FUNCTION_BLOCK FB_Stop
VAR_INPUT
(*È«¾Ö*)
	Mode:DINT;
	PowerState:BOOL;
	CoupleState:DINT;
	(*GapMode*)
	GapStop:BOOL;
	(*BCGapMode*)
	BCGapStop:BOOL;
	(*SingleCarrierMode*)
	TopStop:BOOL;
	BottomStop:BOOL;
	InStop:BOOL;
	OutStop:BOOL;
	(*DebugMode*)
	LeftTopStop:BOOL;
	RightTopStop:BOOL;
	LeftBottomStop:BOOL;
	RightBottomStop:BOOL;
	LeftInStop:BOOL;
	RightInStop:BOOL;
	LeftOutStop:BOOL;
	RightOutStop:BOOL;
END_VAR
VAR_OUTPUT
	FbID:DINT:=1001;
	GapState:DINT;
	GapBusy:BOOL;
	GapDone:BOOL;

	BCGapState:DINT;
	BCGapBusy:BOOL;
	BCGapDone:BOOL;

	TopState:DINT;
	TopBusy:BOOL;
	TopDone:BOOL;
	BottomState:DINT;
	BottomBusy:BOOL;
	BottomDone:BOOL;
	InState:DINT;
	InBusy:BOOL;
	InDone:BOOL;
	OutState:DINT;
	OutBusy:BOOL;
	OutDone:BOOL;

	LeftTopState:DINT;
	LeftTopBusy:BOOL;
	LeftTopDone:BOOL;
	RightTopState:DINT;
	RightTopBusy:BOOL;
	RightTopDone:BOOL;
	LeftBottomState:DINT;
	LeftBottomBusy:BOOL;
	LeftBottomDone:BOOL;
	RightBottomState:DINT;
	RightBottomBusy:BOOL;
	RightBottomDone:BOOL;
	LeftInState:DINT;
	LeftInBusy:BOOL;
	LeftInDone:BOOL;
	RightInState:DINT;
	RightInBusy:BOOL;
	RightInDone:BOOL;
	LeftOutState:DINT;
	LeftOutBusy:BOOL;
	LeftOutDone:BOOL;
	RightOutState:DINT;
	RightOutBusy:BOOL;
	RightOutDone:BOOL;

	Error:BOOL;
	ErrorID:DINT;
END_VAR
VAR
	LeftTop_MC_Stop: MC_Stop;
	LeftBottom_MC_Stop: MC_Stop;
	RightTopLin_MC_Stop: MC_Stop;
	RightBottomLin_MC_Stop: MC_Stop;
	LeftIn_MC_Stop: MC_Stop;
	LeftOut_MC_Stop: MC_Stop;
	RightInLin_MC_Stop: MC_Stop;
	RightOutLin_MC_Stop: MC_Stop;
	fb_ton: TON;
	fb_ton1: TON;
	fb_ton2: TON;
	fb_ton3: TON;
	fb_ton4: TON;
	fb_ton_debug_1:TON;
	fb_ton_debug_2:TON;
	fb_ton_debug_3:TON;
	fb_ton_debug_4:TON;
	fb_ton_debug_5:TON;
	fb_ton_debug_6:TON;
	fb_ton_debug_7:TON;
	fb_ton_debug_8:TON;
	fb_ton_BC: TON;
END_VAR

IF PowerState=1 THEN
	IF Mode=1 AND TopStop THEN
		A_TopStop();
	ELSIF Mode=1 AND BottomStop THEN
		A_BottomStop();
	ELSIF Mode=1 AND InStop THEN
		A_InStop();
	ELSIF Mode=1 AND OutStop THEN
		A_OutStop();
	ELSIF Mode=2 AND LeftTopStop THEN
		A_LeftTopStop();
	ELSIF Mode=2 AND RightTopStop THEN
		A_RightTopStop();
	ELSIF Mode=2 AND LeftBottomStop THEN
		A_LeftBottomStop();
	ELSIF Mode=2 AND RightBottomStop THEN
		A_RightBottomStop();
	ELSIF Mode=2 AND LeftInStop THEN
		A_LeftInStop();
	ELSIF Mode=2 AND RightInStop THEN
		A_RightInStop();
	ELSIF Mode=2 AND LeftOutStop THEN
		A_LeftOutStop();
	ELSIF Mode=2 AND RightOutStop THEN
		A_RightOutStop();
	ELSIF Mode=5 AND BCGapStop THEN
		A_BCGapStop();
	ELSE
		FB_PlcEmergencyStop();
	END_IF
END_IF

ACTION A_BCGapStop:
IF BCGapStop THEN
BCGapBusy:=TRUE;
BCGapDone:=FALSE;
fb_ton_BC(PT:=t#100ms);
A_StopMC();
CASE BCGapState OF
	0:
		IF LeftTop_MC_Stop.Error OR LeftBottom_MC_Stop.Error 
			OR RightTopLin_MC_Stop.Error OR RightBottomLin_MC_Stop.Error
			OR  LeftIn_MC_Stop.Error OR LeftOut_MC_Stop.Error 
			OR RightInLin_MC_Stop.Error OR RightOutLin_MC_Stop.Error THEN
			ErrorID:=1;
			BCGapState:=-100;
			LeftTop_MC_Stop.Execute:=FALSE;
			LeftBottom_MC_Stop.Execute:=FALSE;
			RightTopLin_MC_Stop.Execute:=FALSE;
			RightBottomLin_MC_Stop.Execute:=FALSE;
			LeftIn_MC_Stop.Execute:=FALSE;
			LeftOut_MC_Stop.Execute:=FALSE;
			RightInLin_MC_Stop.Execute:=FALSE;
			RightOutLin_MC_Stop.Execute:=FALSE;
			A_StopMC();
		ELSE
			BCGapState:=1;
		END_IF
	1:
		LeftTop_MC_Stop.Execute:=TRUE;
		LeftBottom_MC_Stop.Execute:=TRUE;
		RightTopLin_MC_Stop.Execute:=TRUE;
		RightBottomLin_MC_Stop.Execute:=TRUE;
		LeftIn_MC_Stop.Execute:=TRUE;
		LeftOut_MC_Stop.Execute:=TRUE;
		RightInLin_MC_Stop.Execute:=TRUE;
		RightOutLin_MC_Stop.Execute:=TRUE;
		fb_ton_BC.IN:=TRUE;
		BCGapState:=2;
	2:
		IF  NOT LeftTop_MC_Stop.Done OR NOT LeftBottom_MC_Stop.Done 
			OR NOT RightTopLin_MC_Stop.Done OR NOT RightBottomLin_MC_Stop.Done
  			OR NOT LeftIn_MC_Stop.Done OR NOT LeftOut_MC_Stop.Done 
			OR NOT RightInLin_MC_Stop.Done OR NOT RightOutLin_MC_Stop.Done THEN
				BCGapState:=2;
		ELSE
			BCGapState:=88;
			LeftTop_MC_Stop.Execute:=FALSE;
			LeftBottom_MC_Stop.Execute:=FALSE;
			RightTopLin_MC_Stop.Execute:=FALSE;
			RightBottomLin_MC_Stop.Execute:=FALSE;			
			LeftIn_MC_Stop.Execute:=FALSE;
			LeftOut_MC_Stop.Execute:=FALSE;
			RightInLin_MC_Stop.Execute:=FALSE;
			RightOutLin_MC_Stop.Execute:=FALSE;
			A_StopMC();
		END_IF

	88:
		BCGapStop:=FALSE;
		BCGapState:=0;
		BCGapBusy:=FALSE;
		BCGapDone:=TRUE;
		Error:=FALSE;
		ErrorID:=0;
		fb_ton_BC.IN:=FALSE;

	-100:
		FB_PlcEmergencyStop();
		BCGapStop:=FALSE;
		BCGapState:=-100;
		BCGapBusy:=FALSE;
		BCGapDone:=FALSE;
		Error:=TRUE;
		LeftTop_MC_Stop.Execute:=FALSE;
		LeftBottom_MC_Stop.Execute:=FALSE;
		RightTopLin_MC_Stop.Execute:=FALSE;
		RightBottomLin_MC_Stop.Execute:=FALSE;			
		LeftIn_MC_Stop.Execute:=FALSE;
		LeftOut_MC_Stop.Execute:=FALSE;
		RightInLin_MC_Stop.Execute:=FALSE;
		RightOutLin_MC_Stop.Execute:=FALSE;
		A_StopMC();
		fb_ton_BC.IN:=FALSE;

END_CASE
END_IF
END_ACTION

ACTION A_BottomStop:
IF BottomStop THEN
BottomBusy:=TRUE;
BottomDone:=FALSE;
fb_ton2(PT:=t#100ms);
A_StopMC();
CASE BottomState OF
	0:
		IF LeftBottom_MC_Stop.Error OR RightBottomLin_MC_Stop.Error THEN
			ErrorID:=1;
			BottomState:=-100;
			LeftBottom_MC_Stop.Execute:=FALSE;
			RightBottomLin_MC_Stop.Execute:=FALSE;
			A_StopMC();
		ELSE
			BottomState:=1;
		END_IF
	1:
		LeftBottom_MC_Stop.Execute:=TRUE;
		RightBottomLin_MC_Stop.Execute:=TRUE;
		fb_ton2.IN:=TRUE;
		BottomState:=2;
	2:
		IF  NOT LeftBottom_MC_Stop.Done OR NOT LeftBottom_MC_Stop.Done THEN
				BottomState:=2;
		ELSE
			BottomState:=88;
			LeftBottom_MC_Stop.Execute:=FALSE;
			RightBottomLin_MC_Stop.Execute:=FALSE;
			A_StopMC();
		END_IF

	88:
		BottomStop:=FALSE;
		BottomState:=0;
		BottomBusy:=FALSE;
		BottomDone:=TRUE;
		Error:=FALSE;
		ErrorID:=0;
		fb_ton2.IN:=FALSE;

	-100:
		FB_PlcEmergencyStop();
		BottomStop:=FALSE;
		BottomState:=-100;
		BottomBusy:=FALSE;
		BottomDone:=FALSE;
		Error:=TRUE;
		LeftBottom_MC_Stop.Execute:=FALSE;
		RightBottomLin_MC_Stop.Execute:=FALSE;
		A_StopMC();
		fb_ton2.IN:=FALSE;

END_CASE
END_IF
END_ACTION

ACTION A_InStop:
IF InStop THEN
InBusy:=TRUE;
InDone:=FALSE;
fb_ton3(PT:=t#100ms);
A_StopMC();
CASE InState OF
	0:
		IF LeftIn_MC_Stop.Error OR RightInLin_MC_Stop.Error THEN
			ErrorID:=1;
			InState:=-100;
			LeftIn_MC_Stop.Execute:=FALSE;
			A_StopMC();
		ELSE
			InState:=1;
		END_IF
	1:
		LeftIn_MC_Stop.Execute:=TRUE;
		RightInLin_MC_Stop.Execute:=TRUE;
		fb_ton3.IN:=TRUE;
		InState:=2;
	2:
		IF  NOT LeftIn_MC_Stop.Done OR NOT RightInLin_MC_Stop.Done THEN
				InState:=2;
		ELSE
			InState:=88;
			LeftIn_MC_Stop.Execute:=FALSE;
			RightInLin_MC_Stop.Execute:=FALSE;
			A_StopMC();
		END_IF

	88:
		InStop:=FALSE;
		InState:=0;
		InBusy:=FALSE;
		InDone:=TRUE;
		Error:=FALSE;
		ErrorID:=0;
		fb_ton3.IN:=FALSE;

	-100:
		FB_PlcEmergencyStop();
		InStop:=FALSE;
		InState:=-100;
		InBusy:=FALSE;
		InDone:=FALSE;
		Error:=TRUE;
		LeftIn_MC_Stop.Execute:=FALSE;
		RightInLin_MC_Stop.Execute:=FALSE;
		A_StopMC();
		fb_ton3.IN:=FALSE;

END_CASE
END_IF
END_ACTION

ACTION A_LeftBottomStop:
IF LeftBottomStop THEN
LeftBottomBusy:=TRUE;
LeftBottomDone:=FALSE;
fb_ton_debug_3(PT:=t#100ms);
A_StopMC();
CASE LeftBottomState OF
	0:
		IF LeftBottom_MC_Stop.Error THEN
			ErrorID:=41;
			LeftBottomState:=-100;
			LeftBottom_MC_Stop.Execute:=FALSE;
			A_StopMC();
		ELSE
			LeftBottomState:=1;
		END_IF
	1:
		LeftBottom_MC_Stop.Execute:=TRUE;
		fb_ton_debug_3.IN:=TRUE;
		LeftBottomState:=2;
	2:
		IF  NOT LeftBottom_MC_Stop.Done THEN
				LeftBottomState:=2;
		ELSE
			LeftBottomState:=88;
			LeftBottom_MC_Stop.Execute:=FALSE;
			A_StopMC();
		END_IF

	88:
		LeftBottomStop:=FALSE;
		LeftBottomState:=0;
		LeftBottomBusy:=FALSE;
		LeftBottomDone:=TRUE;
		Error:=FALSE;
		ErrorID:=0;
		fb_ton_debug_3.IN:=FALSE;

	-100:
		FB_PlcEmergencyStop();
		LeftBottomStop:=FALSE;
		LeftBottomState:=-100;
		LeftBottomBusy:=FALSE;
		LeftBottomDone:=FALSE;
		Error:=TRUE;
		LeftBottom_MC_Stop.Execute:=FALSE;
		A_StopMC();
		fb_ton_debug_3.IN:=FALSE;

END_CASE
END_IF
END_ACTION

ACTION A_LeftInStop:
IF LeftInStop THEN
LeftInBusy:=TRUE;
LeftInDone:=FALSE;
fb_ton_debug_4(PT:=t#100ms);
A_StopMC();
CASE LeftInState OF
	0:
		IF LeftIn_MC_Stop.Error THEN
			ErrorID:=41;
			LeftInState:=-100;
			LeftIn_MC_Stop.Execute:=FALSE;
			A_StopMC();
		ELSE
			LeftInState:=1;
		END_IF
	1:
		LeftIn_MC_Stop.Execute:=TRUE;
		fb_ton_debug_4.IN:=TRUE;
		LeftInState:=2;
	2:
		IF  NOT LeftIn_MC_Stop.Done THEN
				LeftInState:=2;
		ELSE
			LeftInState:=88;
			LeftIn_MC_Stop.Execute:=FALSE;
			A_StopMC();
		END_IF

	88:
		LeftInStop:=FALSE;
		LeftInState:=0;
		LeftInBusy:=FALSE;
		LeftInDone:=TRUE;
		Error:=FALSE;
		ErrorID:=0;
		fb_ton_debug_4.IN:=FALSE;

	-100:
		FB_PlcEmergencyStop();
		LeftInStop:=FALSE;
		LeftInState:=-100;
		LeftInBusy:=FALSE;
		LeftInDone:=FALSE;
		Error:=TRUE;
		LeftIn_MC_Stop.Execute:=FALSE;
		A_StopMC();
		fb_ton_debug_4.IN:=FALSE;

END_CASE
END_IF
END_ACTION

ACTION A_LeftOutStop:
IF LeftOutStop THEN
LeftOutBusy:=TRUE;
LeftOutDone:=FALSE;
fb_ton_debug_7(PT:=t#100ms);
A_StopMC();
CASE LeftOutState OF
	0:
		IF LeftOut_MC_Stop.Error THEN
			ErrorID:=41;
			LeftOutState:=-100;
			LeftOut_MC_Stop.Execute:=FALSE;
			A_StopMC();
		ELSE
			LeftOutState:=1;
		END_IF
	1:
		LeftOut_MC_Stop.Execute:=TRUE;
		fb_ton_debug_7.IN:=TRUE;
		LeftOutState:=2;
	2:
		IF  NOT LeftOut_MC_Stop.Done THEN
				LeftOutState:=2;
		ELSE
			LeftOutState:=88;
			LeftOut_MC_Stop.Execute:=FALSE;
			A_StopMC();
		END_IF

	88:
		LeftOutStop:=FALSE;
		LeftOutState:=0;
		LeftOutBusy:=FALSE;
		LeftOutDone:=TRUE;
		Error:=FALSE;
		ErrorID:=0;
		fb_ton_debug_7.IN:=FALSE;

	-100:
		FB_PlcEmergencyStop();
		LeftOutStop:=FALSE;
		LeftOutState:=-100;
		LeftOutBusy:=FALSE;
		LeftOutDone:=FALSE;
		Error:=TRUE;
		LeftOut_MC_Stop.Execute:=FALSE;
		A_StopMC();
		fb_ton_debug_7.IN:=FALSE;

END_CASE
END_IF
END_ACTION

ACTION A_LeftTopStop:
IF LeftTopStop THEN
LeftTopBusy:=TRUE;
LeftTopDone:=FALSE;
fb_ton_debug_1(PT:=t#100ms);
A_StopMC();
CASE LeftTopState OF
	0:
		IF LeftTop_MC_Stop.Error THEN
			ErrorID:=41;
			LeftTopState:=-100;
			LeftTop_MC_Stop.Execute:=FALSE;
			A_StopMC();
		ELSE
			LeftTopState:=1;
		END_IF
	1:
		LeftTop_MC_Stop.Execute:=TRUE;
		fb_ton_debug_1.IN:=TRUE;
		LeftTopState:=2;
	2:
		IF  NOT LeftTop_MC_Stop.Done THEN
				LeftTopState:=2;
		ELSE
			LeftTopState:=88;
			LeftTop_MC_Stop.Execute:=FALSE;
			A_StopMC();
		END_IF

	88:
		LeftTopStop:=FALSE;
		LeftTopState:=0;
		LeftTopBusy:=FALSE;
		LeftTopDone:=TRUE;
		Error:=FALSE;
		ErrorID:=0;
		fb_ton_debug_1.IN:=FALSE;

	-100:
		FB_PlcEmergencyStop();
		LeftTopStop:=FALSE;
		LeftTopState:=-100;
		LeftTopBusy:=FALSE;
		LeftTopDone:=FALSE;
		Error:=TRUE;
		LeftTop_MC_Stop.Execute:=FALSE;
		A_StopMC();
		fb_ton_debug_1.IN:=FALSE;

END_CASE
END_IF
END_ACTION

ACTION A_OutStop:
IF OutStop THEN
OutBusy:=TRUE;
OutDone:=FALSE;
fb_ton4(PT:=T#100MS);
A_StopMC();
CASE OutState OF
	0:
		IF LeftOut_MC_Stop.Error OR RightOutLin_MC_Stop.Error THEN
			ErrorID:=1;
			OutState:=-100;
			LeftOut_MC_Stop.Execute:=FALSE;
			RightOutLin_MC_Stop.Execute:=FALSE;
			A_StopMC();
		ELSE
			OutState:=1;
		END_IF
	1:
		LeftOut_MC_Stop.Execute:=TRUE;
		RightOutLin_MC_Stop.Execute:=TRUE;
		fb_ton4.IN:=TRUE;
		OutState:=2;
	2:
		IF  NOT LeftOut_MC_Stop.Done OR NOT LeftOut_MC_Stop.Done THEN
				OutState:=2;
		ELSE
			OutState:=88;
			LeftOut_MC_Stop.Execute:=FALSE;
			RightOutLin_MC_Stop.Execute:=FALSE;
			A_StopMC();
		END_IF

	88:
		OutStop:=FALSE;
		OutState:=0;
		OutBusy:=FALSE;
		OutDone:=TRUE;
		Error:=FALSE;
		ErrorID:=0;
		fb_ton4.IN:=FALSE;

	-100:
		FB_PlcEmergencyStop();
		OutStop:=FALSE;
		OutState:=-100;
		OutBusy:=FALSE;
		OutDone:=FALSE;
		Error:=TRUE;
		LeftOut_MC_Stop.Execute:=FALSE;
		RightOutLin_MC_Stop.Execute:=FALSE;
		A_StopMC();
		fb_ton4.IN:=FALSE;

END_CASE
END_IF
END_ACTION

ACTION A_RightBottomStop:
IF RightBottomStop THEN
RightBottomBusy:=TRUE;
RightBottomDone:=FALSE;
fb_ton_debug_4(PT:=t#100ms);
A_StopMC();
CASE RightBottomState OF
	0:
		IF RightBottomLin_MC_Stop.Error THEN
			ErrorID:=41;
			RightBottomState:=-100;
			RightBottomLin_MC_Stop.Execute:=FALSE;
			A_StopMC();
		ELSE
			RightBottomState:=1;
		END_IF
	1:
		RightBottomLin_MC_Stop.Execute:=TRUE;
		fb_ton_debug_4.IN:=TRUE;
		RightBottomState:=2;
	2:
		IF  NOT RightBottomLin_MC_Stop.Done THEN
				RightBottomState:=2;
		ELSE
			RightBottomState:=88;
			RightBottomLin_MC_Stop.Execute:=FALSE;
			A_StopMC();
		END_IF

	88:
		RightBottomStop:=FALSE;
		RightBottomState:=0;
		RightBottomBusy:=FALSE;
		RightBottomDone:=TRUE;
		Error:=FALSE;
		ErrorID:=0;
		fb_ton_debug_4.IN:=FALSE;

	-100:
		FB_PlcEmergencyStop();
		RightBottomStop:=FALSE;
		RightBottomState:=-100;
		RightBottomBusy:=FALSE;
		RightBottomDone:=FALSE;
		Error:=TRUE;
		RightBottomLin_MC_Stop.Execute:=FALSE;
		A_StopMC();
		fb_ton_debug_4.IN:=FALSE;

END_CASE
END_IF
END_ACTION

ACTION A_RightInStop:
IF RightInStop THEN
RightInBusy:=TRUE;
RightInDone:=FALSE;
fb_ton_debug_6(PT:=t#100ms);
A_StopMC();
CASE RightInState OF
	0:
		IF RightInLin_MC_Stop.Error THEN
			ErrorID:=41;
			RightInState:=-100;
			RightInLin_MC_Stop.Execute:=FALSE;
			A_StopMC();
		ELSE
			RightInState:=1;
		END_IF
	1:
		RightInLin_MC_Stop.Execute:=TRUE;
		fb_ton_debug_6.IN:=TRUE;
		RightInState:=2;
	2:
		IF  NOT RightInLin_MC_Stop.Done THEN
				RightInState:=2;
		ELSE
			RightInState:=88;
			RightInLin_MC_Stop.Execute:=FALSE;
			A_StopMC();
		END_IF

	88:
		RightInStop:=FALSE;
		RightInState:=0;
		RightInBusy:=FALSE;
		RightInDone:=TRUE;
		Error:=FALSE;
		ErrorID:=0;
		fb_ton_debug_6.IN:=FALSE;

	-100:
		FB_PlcEmergencyStop();
		RightInStop:=FALSE;
		RightInState:=-100;
		RightInBusy:=FALSE;
		RightInDone:=FALSE;
		Error:=TRUE;
		RightInLin_MC_Stop.Execute:=FALSE;
		A_StopMC();
		fb_ton_debug_6.IN:=FALSE;

END_CASE
END_IF
END_ACTION

ACTION A_RightOutStop:
IF RightOutStop THEN
RightOutBusy:=TRUE;
RightOutDone:=FALSE;
fb_ton_debug_8(PT:=t#100ms);
A_StopMC();
CASE RightOutState OF
	0:
		IF RightOutLin_MC_Stop.Error THEN
			ErrorID:=41;
			RightOutState:=-100;
			RightOutLin_MC_Stop.Execute:=FALSE;
			A_StopMC();
		ELSE
			RightOutState:=1;
		END_IF
	1:
		RightOutLin_MC_Stop.Execute:=TRUE;
		fb_ton_debug_8.IN:=TRUE;
		RightOutState:=2;
	2:
		IF  NOT RightOutLin_MC_Stop.Done THEN
				RightOutState:=2;
		ELSE
			RightOutState:=88;
			RightOutLin_MC_Stop.Execute:=FALSE;
			A_StopMC();
		END_IF

	88:
		RightOutStop:=FALSE;
		RightOutState:=0;
		RightOutBusy:=FALSE;
		RightOutDone:=TRUE;
		Error:=FALSE;
		ErrorID:=0;
		fb_ton_debug_8.IN:=FALSE;

	-100:
		FB_PlcEmergencyStop();
		RightOutStop:=FALSE;
		RightOutState:=-100;
		RightOutBusy:=FALSE;
		RightOutDone:=FALSE;
		Error:=TRUE;
		RightOutLin_MC_Stop.Execute:=FALSE;
		A_StopMC();
		fb_ton_debug_8.IN:=FALSE;

END_CASE
END_IF
END_ACTION

ACTION A_RightTopStop:
IF RightTopStop THEN
RightTopBusy:=TRUE;
RightTopDone:=FALSE;
fb_ton_debug_2(PT:=t#100ms);
A_StopMC();
CASE RightTopState OF
	0:
		IF RightTopLin_MC_Stop.Error THEN
			ErrorID:=41;
			RightTopState:=-100;
			RightTopLin_MC_Stop.Execute:=FALSE;
			A_StopMC();
		ELSE
			RightTopState:=1;
		END_IF
	1:
		RightTopLin_MC_Stop.Execute:=TRUE;
		fb_ton_debug_2.IN:=TRUE;
		RightTopState:=2;
	2:
		IF  NOT RightTopLin_MC_Stop.Done THEN
				RightTopState:=2;
		ELSE
			RightTopState:=88;
			RightTopLin_MC_Stop.Execute:=FALSE;
			A_StopMC();
		END_IF

	88:
		RightTopStop:=FALSE;
		RightTopState:=0;
		RightTopBusy:=FALSE;
		RightTopDone:=TRUE;
		Error:=FALSE;
		ErrorID:=0;
		fb_ton_debug_2.IN:=FALSE;

	-100:
		FB_PlcEmergencyStop();
		RightTopStop:=FALSE;
		RightTopState:=-100;
		RightTopBusy:=FALSE;
		RightTopDone:=FALSE;
		Error:=TRUE;
		RightTopLin_MC_Stop.Execute:=FALSE;
		A_StopMC();
		fb_ton_debug_2.IN:=FALSE;

END_CASE
END_IF
END_ACTION

ACTION A_StopMC:
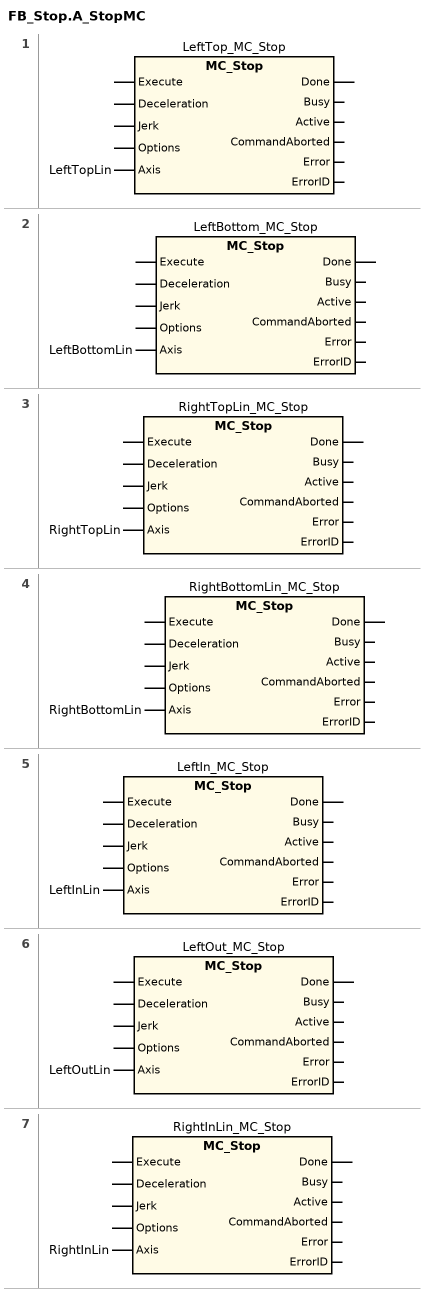
// NETWORK 1
LeftTop_MC_Stop(Axis := LeftTopLin); // MC_Stop

// NETWORK 2
LeftBottom_MC_Stop(Axis := LeftBottomLin); // MC_Stop

// NETWORK 3
RightTopLin_MC_Stop(Axis := RightTopLin); // MC_Stop

// NETWORK 4
RightBottomLin_MC_Stop(Axis := RightBottomLin); // MC_Stop

// NETWORK 5
LeftIn_MC_Stop(Axis := LeftInLin); // MC_Stop

// NETWORK 6
LeftOut_MC_Stop(Axis := LeftOutLin); // MC_Stop

// NETWORK 7
RightInLin_MC_Stop(Axis := RightInLin); // MC_Stop

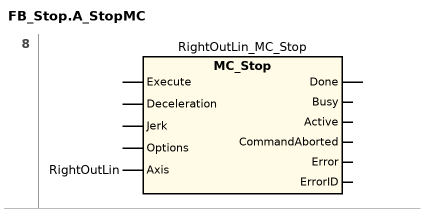
// NETWORK 8
RightOutLin_MC_Stop(Axis := RightOutLin); // MC_Stop
END_ACTION

ACTION A_TopStop:
IF TopStop THEN
TopBusy:=TRUE;
TopDone:=FALSE;
fb_ton1(PT:=t#100ms);
A_StopMC();
CASE TopState OF
	0:
		IF LeftTop_MC_Stop.Error OR RightTopLin_MC_Stop.Error THEN
			ErrorID:=1;
			TopState:=-100;
			LeftTop_MC_Stop.Execute:=FALSE;
			A_StopMC();
		ELSE
			TopState:=1;
		END_IF
	1:
		LeftTop_MC_Stop.Execute:=TRUE;
		RightTopLin_MC_Stop.Execute:=TRUE;
		fb_ton1.IN:=TRUE;
		TopState:=2;
	2:
		IF  NOT LeftTop_MC_Stop.Done OR NOT RightTopLin_MC_Stop.Done THEN
				TopState:=2;
		ELSE
			TopState:=88;
			LeftTop_MC_Stop.Execute:=FALSE;
			RightTopLin_MC_Stop.Execute:=FALSE;
			A_StopMC();
		END_IF

	88:
		TopStop:=FALSE;
		TopState:=0;
		TopBusy:=FALSE;
		TopDone:=TRUE;
		Error:=FALSE;
		ErrorID:=0;
		fb_ton1.IN:=FALSE;

	-100:
		FB_PlcEmergencyStop();
		TopStop:=FALSE;
		TopState:=-100;
		TopBusy:=FALSE;
		TopDone:=FALSE;
		Error:=TRUE;
		LeftTop_MC_Stop.Execute:=FALSE;
		RightTopLin_MC_Stop.Execute:=FALSE;
		A_StopMC();
		fb_ton1.IN:=FALSE;

END_CASE
END_IF
END_ACTION

END_FUNCTION_BLOCK

(* stored: Version 1.1.0.1, ProductVersion 3.1.4024.6
   POU FB_Stop: Id {3e354bcb-4e4f-4b34-9851-51b9542d0760}, SpecialFunc None
   Folder Debug: Id {104af77a-ff55-4e7d-ae89-0786c90d6988}
   Folder SingleCarrier: Id {5f2d3879-30be-4d08-a393-873fa14fb1eb}
   Folder UserMode: Id {c0a55f07-0d1e-4846-a7f6-2b5ce6b13305}
   Action A_BCGapStop: Id {09d39807-0cc9-4816-a94c-73c13504c1f7}
   Action A_BottomStop: Id {3e5d2212-d55d-4178-a1aa-10c2e89eefb4}
   Action A_InStop: Id {f06e74fd-318c-415b-ac2b-adabc6072b86}
   Action A_LeftBottomStop: Id {cab19fe7-18d8-423d-84e7-b2a63e643950}
   Action A_LeftInStop: Id {f91b09e3-f669-4f08-abb4-4e66bddd882d}
   Action A_LeftOutStop: Id {c9624617-5b4c-46c3-afa1-8314afa61125}
   Action A_LeftTopStop: Id {2b524d72-b139-4ac0-8fb1-7a7578319dea}
   Action A_OutStop: Id {7cd401e6-bd12-4ae4-a499-be9296d9c5d9}
   Action A_RightBottomStop: Id {e95ff139-ca76-4481-866d-edf0363d8b42}
   Action A_RightInStop: Id {2cda54c4-d20f-4c2e-a0eb-d55ad846c492}
   Action A_RightOutStop: Id {81ad3fea-d849-44a0-8cfd-690db5e1ec0a}
   Action A_RightTopStop: Id {81452b6a-45dc-414d-8661-6860831ad67d}
   Action A_StopMC: Id {b171a3f0-94b4-4ac2-92c0-8ca964cc4005}
   Action A_TopStop: Id {35574051-d064-41d9-8c90-d1d9b62d4922} *)
